// TIA Portal project "Projeto Final Partiu bar Parte 4 - A terra e o tempo" (V11)

(* hardware
DEVICE "HMI_1"  TP 177B 6" PN/DP
   slot 0: "HMI"  HMI  6AV6642-0BA01-1AX1  11.0.0
   slot 1: "HMI_RT_1"  TP 177B 6" PN/DP  6AV6642-0BA01-1AX1  11.0.0
   slot 5: "IE_CP_1"  PROFINET interface  IE_CP  V7.1.0
      slot 1: "PROFINET_Interface_1"  HMI IE SUBMODULE
         slot 1: "PORT_1"  HMI IE PORTMODULE 1  1.0.0.0
   slot 7: "MPI/DP_CP_1"  HMI MPIDP  MPI-DP_CP  1.0.0.0
DEVICE "ET 200S station_1"  ET200S-Station
   slot 0: "Rack"  Rail
   slot 2: "PLC_1"  IM151-8 F-CPU  6ES7 151-8FB01-0AB0  V3.2
      slot 1: "PROFINET interface_1"  PN-IO
         slot 1: "Port_1"  Port
         slot 2: "Port_2"  Port
         slot 3: "Port_3"  Port
   slot 4: "PM-E DC24V /8A RO_1"  6ES7 138-4CA80-0AB0
   slot 5: "4DI x 24VDC HF_1"  4DI DC24V HF  6ES7 131-4BD01-0AB0
   slot 6: "4DI x 24VDC HF_2"  4DI DC24V HF  6ES7 131-4BD01-0AB0
   slot 7: "4DI x 24VDC HF_3"  4DI DC24V HF  6ES7 131-4BD01-0AB0
   slot 8: "4DI x 24VDC HF_4"  4DI DC24V HF  6ES7 131-4BD01-0AB0
   slot 9: "4DI x 24VDC HF_5"  4DI DC24V HF  6ES7 131-4BD01-0AB0
   slot 10: "4DO x 24VDC / 0.5A HF_1"  4DO DC24V/0.5A HF  6ES7 132-4BD00-0AB0
   slot 11: "4DO x 24VDC / 0.5A HF_2"  4DO DC24V/0.5A HF  6ES7 132-4BD00-0AB0
   slot 12: "PM-E DC24V /8A RO_2"  6ES7 138-4CA80-0AB0
   slot 13: "4DO x 24VDC / 0.5A HF_3"  4DO DC24V/0.5A HF  6ES7 132-4BD00-0AB0
   slot 14: "4DO x 24VDC / 0.5A HF_4"  4DO DC24V/0.5A HF  6ES7 132-4BD00-0AB0
   slot 15: "4DO x 24VDC / 0.5A HF_5"  4DO DC24V/0.5A HF  6ES7 132-4BD00-0AB0
   slot 16: "2AI x U HF_1"  2AI U HF  6ES7 134-4LB02-0AB0
   slot 17: "2AI x U HF_2"  2AI U HF  6ES7 134-4LB02-0AB0
   slot 18: "2AO x U HF_1"  2AO U HF  6ES7 135-4LB02-0AB0
   slot 19: "1 Count 24V_1"  1 COUNT 24V/100 kHz C/F/M/W  6ES7 138-4DA04-0AB0  V2.0
   slot 20: "4SI IO link_1"  4SI IO-Link  6ES7 138-4GA50-0AB0
*)

// ===== PLC "PLC_1"  IM151-8 F-CPU =====

VAR_GLOBAL   // PLC tag table "Default tag table"
   "e0" AT %M0.0 : Bool;   // Estado 0
   "e10" AT %M0.1 : Bool;   // Estado 1.0
   "start" AT %I2.0 : Bool;   // Inicia o sistema
   "e20" AT %M0.2 : Bool;   // Estado 2.0
   "e4" AT %M0.4 : Bool;   // Estado 4
   "e30" AT %M0.3 : Bool;   // Estado 3.0
   "e11" AT %M0.5 : Bool;   // Estado 1.1
   "e21" AT %M0.6 : Bool;   // Estado 2.1
   "vcv" AT %Q6.3 : Bool;   // Valvula cerveja verde
   "vcm" AT %Q6.2 : Bool;   // Valvula cerveja maturada
   "vfr" AT %Q7.0 : Bool;   // Valvula fluido refrigerante
   "sbm" AT %I1.0 : Bool;   // Sensor de nivel baixo maturador
   "sbf" AT %I1.1 : Bool;   // Sensor de nivel baixo filtro
   "iniciar" AT %M6.2 : Bool;   // Botao iniciar
   "T.P" AT %IW448 : Int;   // Sinal de temperatura
   "Tdig" AT %MD1 : Real;   // Temperatura do maturador
   "Tscale" AT %MW3 : Int;   // Sinal de temperatura digital
   "False" AT %M6.0 : Bool;   // Variavel auxiliar = 0
   "Error" AT %MW7 : Word;   // Variavel auxiliar
   "homming" AT %M6.1 : Bool;   // Modo homming
   "pap" AT %M6.3 : Bool;   // Modo passo a passo
   "passo" AT %M6.4 : Bool;   // Botao de passo
   "emergencia" AT %M6.5 : Bool;   // Modo de emergencia
   "alarme" AT %M6.6 : Bool;   // Estado de Alarme
   "alarmeFiltro" AT %M5.0 : Bool;   // Alarme por tempo do filtro
   "alarmeRefrig" AT %M5.1 : Bool;   // Alarme por tempo do Refrigerante
   "ResetAlarm" AT %M5.2 : Bool;   // Reseta alarme
   "TrataAlarme" AT %M5.3 : Bool;
   "alarmeCond" AT %M5.4 : Bool;   // Condicao de alarme
   "em0" AT %M9.0 : Bool;   // Estado de emergencia 0
   "em10" AT %M9.1 : Bool;   // Estado de emergencia 1.0
   "em20" AT %M9.2 : Bool;   // Estado de emergencia 2.0
   "em30" AT %M9.3 : Bool;   // Estado de emergencia 3.0
   "em4" AT %M9.4 : Bool;   // Estado de emergencia 4
   "em11" AT %M9.5 : Bool;   // Estado de emergencia 1.1
   "em21" AT %M9.6 : Bool;   // Estado de emergencia 2.1
   "auto" AT %M9.7 : Bool;   // Modo automatico
   "vtd" AT %Q7.1 : Bool;   // Valvula de terra diatomacea
   "vr" AT %Q7.2 : Bool;   // Valvula de residuos
   "tenchimento" AT %M5.5 : Bool;   // Tempo de enchimento atingido
   "tmaturacao" AT %M5.6 : Bool;   // Tempo de maturacao atingido
   "alarmeMat" AT %M5.7 : Bool;   // Alarme por tempo do maturador
   "alarmeTemp" AT %M6.7 : Bool;   // Alarme temperatura
   "homeCount" AT %MW2 : Int;   // Contador de ciclos
   "cleanMat" AT %M10.0 : Bool;   // Botao Limpeza Maturador
   "cleanFilt" AT %M10.1 : Bool;   // Botao Limpeza Filtro
   "em6" AT %M10.2 : Bool;   // Estado Limpeza Maturador
   "em7" AT %M10.3 : Bool;   // Estado Limpeza Filtro
END_VAR

ORGANIZATION_BLOCK "Main"   // OB1, LAD
TITLE = "Main Program Sweep (Cycle)"
{ S7_Optimized_Access := 'FALSE' }
VERSION : 0.1
   VAR_TEMP
      OB1_EV_CLASS : Byte;   // Bits 0-3 = 1 (Coming event), Bits 4-7 = 1 (Event class 1)
      OB1_SCAN_1 : Byte;   // 1 (Cold restart scan 1 of OB 1), 3 (Scan 2-n of OB 1)
      OB1_PRIORITY : Byte;   // Priority of OB Execution
      OB1_OB_NUMBR : Byte;   // 1 (Organization block 1, OB1)
      OB1_RESERVED_1 : Byte;   // Reserved for system
      OB1_RESERVED_2 : Byte;   // Reserved for system
      OB1_PREV_CYCLE : Int;   // Cycle time of previous OB1 scan (milliseconds)
      OB1_MIN_CYCLE : Int;   // Minimum cycle time of OB1 (milliseconds)
      OB1_MAX_CYCLE : Int;   // Maximum cycle time of OB1 (milliseconds)
      OB1_DATE_TIME : Date_And_Time;   // Date and time OB1 started
   END_VAR
BEGIN
END_ORGANIZATION_BLOCK